PROGRAM WriteAnalogOutputCurrent
VAR
	temp: REAL;
END_VAR

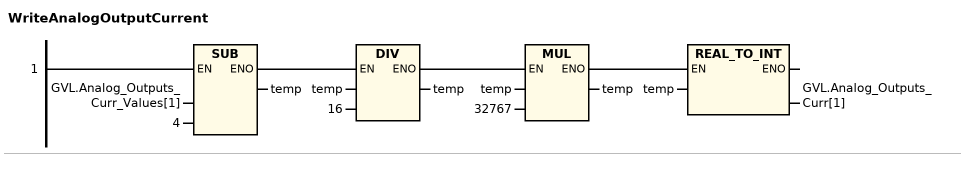
// NETWORK 1
temp := GVL.Analog_Outputs_Curr_Values[1] - 4;
temp := temp / 16;
temp := temp * 32767;
GVL.Analog_Outputs_Curr[1] := REAL_TO_INT(temp);

END_PROGRAM

(* stored: Version 1.1.0.1, ProductVersion 3.1.4024.12
   POU WriteAnalogOutputCurrent: Id {c8ebc1bf-e381-4300-b006-ac846a16ec5a}, SpecialFunc None *)
